(*Spectroscopy scanning Mode*)
IF IsSSMotionMode THEN
	SSMotionMode:=TRUE;
	RegularMotionMode:=FALSE;
ELSE
	SSMotionMode:=FALSE;
	RegularMotionMode:=TRUE;
END_IF
IF	SSMotionMode AND NOT RegularMotionMode THEN
	A_SpectroscopyScanningMotion();
END_IF

(*CheckInputPosVelo*)
A_CheckInputPosVelo();
(*检查光栅读数是否在范围内*)
A_CheckLinearEncoder();

ACTION A_CheckCoupleStatus:
IF NOT btn_PowerOff THEN
	IF st_Power=1 AND st_Couple<>0THEN
		Error:=TRUE;
		ErrorID:=501;
		LeftTopLinMoveIndicator:=0;
		RightTopLinMoveIndicator:=0;
		LeftBottomLinMoveIndicator:=0;
		RightBottomLinMoveIndicator:=0;
		FB_PlcEmergencyStop();
		LED_Error:=TRUE;
		ErrorDescription:='couple stutas error';
	END_IF
END_IF
END_ACTION

ACTION A_CheckInputPosVelo:
//gap posiion
IF UserGapPositionNew<min_UserGapPositionNew OR UserGapPositionNew>max_UserGapPositionNew THEN
	inRange_UserGapPositionNew:=FALSE;
END_IF
IF UserGapPositionNew>=min_UserGapPositionNew AND UserGapPositionNew<=max_UserGapPositionNew THEN
	inRange_UserGapPositionNew:=TRUE;
END_IF
//gap velocity
IF UserGapVelocityNew<min_UserGapVelocityNew OR UserGapVelocityNew>max_UserGapVelocityNew THEN
	inRange_UserGapVelocityNew:=FALSE;
END_IF
IF UserGapVelocityNew>=min_UserGapVelocityNew AND UserGapVelocityNew<=max_UserGapVelocityNew THEN
	inRange_UserGapVelocityNew:=TRUE;
END_IF
//taper position
IF UserTaperPositionNew<min_UserTaperPositionNew OR UserTaperPositionNew>max_UserTaperPositionNew THEN
	inRange_UserTaperPositionNew:=FALSE;
END_IF
IF UserTaperPositionNew>=min_UserTaperPositionNew AND UserTaperPositionNew<=max_UserTaperPositionNew THEN
	inRange_UserTaperPositionNew:=TRUE;
END_IF
//taper velocity
IF UserTaperVelocityNew<min_UserTaperVelocityNew OR UserTaperVelocityNew>max_UserTaperVelocityNew THEN
	inRange_UserTaperVelocityNew:=FALSE;
END_IF
IF UserTaperVelocityNew>=min_UserTaperVelocityNew AND UserTaperVelocityNew<=max_UserTaperVelocityNew THEN
	inRange_UserTaperVelocityNew:=TRUE;
END_IF
//SS Mode
IF SS_StepSize<min_SS_StepSize OR SS_StepSize>max_SS_StepSize THEN
	inRange_SS_StepSize:=FALSE;
END_IF
IF SS_StepSize>=min_SS_StepSize AND SS_StepSize<=max_SS_StepSize THEN
	inRange_SS_StepSize:=TRUE;
END_IF
IF SS_StepNumber<min_SS_StepNumber OR SS_StepNumber>max_SS_StepNumber THEN
	inRange_SS_StepNumber:=FALSE;
END_IF
IF SS_StepNumber>=min_SS_StepNumber AND SS_StepNumber<=max_SS_StepNumber THEN
	inRange_SS_StepNumber:=TRUE;
END_IF
IF SS_StepVelocity<min_SS_StepVelocity OR SS_StepVelocity>max_SS_StepVelocity THEN
	inRange_SS_StepVelocity:=FALSE;
END_IF
IF SS_StepVelocity>=min_SS_StepVelocity AND SS_StepVelocity<=max_SS_StepVelocity THEN
	inRange_SS_StepVelocity:=TRUE;
END_IF
IF StepEachTime_ms<min_StepEachTime_ms OR StepEachTime_ms>max_StepEachTime_ms THEN
	inRange_StepEachTime_ms:=FALSE;
END_IF
IF StepEachTime_ms>=min_StepEachTime_ms AND StepEachTime_ms<=max_StepEachTime_ms THEN
	inRange_StepEachTime_ms:=TRUE;
END_IF
END_ACTION

ACTION A_CheckLinearEncoder:
//如果没有使用光栅、或者光栅参数没设置好，则不检查光栅位置
IF NOT USELinearEncoder OR NOT PositionBiasDone THEN
	RETURN;
END_IF
IF Pos_LeftTopLin <=0 THEN
	ErrorID:=1101;
	Error:=TRUE;
	ErrorDescription:='Pos_LeftTopLin <=0';
	FB_PlcEmergencyStop();
	LED_Error:=TRUE;
END_IF
IF Pos_RightTopLin <=0 THEN
	ErrorID:=1102;
	Error:=TRUE;
	ErrorDescription:='Pos_RightTopLin <=0';
	FB_PlcEmergencyStop();
	LED_Error:=TRUE;
END_IF
IF Pos_LeftBottomLin <=0 THEN
	ErrorID:=1103;
	Error:=TRUE;
	ErrorDescription:='Pos_LeftBottomLin <=0';
	FB_PlcEmergencyStop();
	LED_Error:=TRUE;
END_IF
IF Pos_RightBottomLin <=0 THEN
	ErrorID:=1104;
	Error:=TRUE;
	ErrorDescription:='Pos_RightBottomLin <=0';
	FB_PlcEmergencyStop();
	LED_Error:=TRUE;
END_IF
//
IF Pos_LeftTopLin >UserMode.max_UserGapPositionNew/2 THEN
	ErrorID:=1105;
	Error:=TRUE;
	ErrorDescription:='Pos_LeftTopLin >UserMode.max_UserGapPositionNew';
	FB_PlcEmergencyStop();
	LED_Error:=TRUE;
END_IF
IF Pos_RightTopLin >UserMode.max_UserGapPositionNew/2 THEN
	ErrorID:=1106;
	Error:=TRUE;
	ErrorDescription:='Pos_RightTopLin>UserMode.max_UserGapPositionNew';
	FB_PlcEmergencyStop();
	LED_Error:=TRUE;
END_IF
IF Pos_LeftBottomLin >UserMode.max_UserGapPositionNew/2 THEN
	ErrorID:=1107;
	Error:=TRUE;
	ErrorDescription:='Pos_LeftBottomLin >UserMode.max_UserGapPositionNew';
	FB_PlcEmergencyStop();
	LED_Error:=TRUE;
END_IF
IF Pos_RightBottomLin >UserMode.max_UserGapPositionNew/2 THEN
	ErrorID:=1108;
	Error:=TRUE;
	ErrorDescription:='Pos_RightBottomLin >UserMode.max_UserGapPositionNew';
	FB_PlcEmergencyStop();
	LED_Error:=TRUE;
END_IF

//
IF Pos_LeftTopLin <UserMode.min_UserGapPositionNew/2 THEN
	ErrorID:=1109;
	Error:=TRUE;
	ErrorDescription:='Pos_LeftTopLin <UserMode.min_UserGapPositionNew/2';
	FB_PlcEmergencyStop();
	LED_Error:=TRUE;
END_IF
IF Pos_RightTopLin <UserMode.min_UserGapPositionNew/2 THEN
	ErrorID:=1110;
	Error:=TRUE;
	ErrorDescription:='Pos_RightTopLin<UserMode.min_UserGapPositionNew/2';
	FB_PlcEmergencyStop();
	LED_Error:=TRUE;
END_IF
IF Pos_LeftBottomLin <UserMode.min_UserGapPositionNew/2 THEN
	ErrorID:=1111;
	Error:=TRUE;
	ErrorDescription:='Pos_LeftBottomLin <UserMode.min_UserGapPositionNew';
	FB_PlcEmergencyStop();
	LED_Error:=TRUE;
END_IF
IF Pos_RightBottomLin <UserMode.min_UserGapPositionNew/2 THEN
	ErrorID:=1112;
	Error:=TRUE;
	ErrorDescription:='Pos_RightBottomLin <UserMode.min_UserGapPositionNew';
	FB_PlcEmergencyStop();
	LED_Error:=TRUE;
END_IF
END_ACTION

ACTION A_InitCompensationData:
(*补偿开始*)
IF USE_SingleAxis_Compensation THEN
	//
	//1.目标位置解算
	//
	(*通过补偿表解算四轴目标位置*)
	//左轴位置由Gap定，右轴位置由右gap定。右gap值=左gap+taper。taper模式和非taper模式一样，非taper模式只是一种特例存在
	//左轴目标位置解算
	IF NOT TaperOrNot THEN
		UserTaperPositionNew:=0;
		UserTaperPositionDisplay:=0;
	END_IF
	UserRightGapPositionNew:=UserGapPositionNew+UserTaperPositionNew;
	//左轴目标位置解算
	FOR	i:= 1 TO 17 DO
			IF UserGapPositionNew/2<M_Compensation[i+1].Encoder AND UserGapPositionNew/2>=M_Compensation[i].Encoder THEN
				IF i<>18 THEN
					LeftTopLinPositionNew:=(((UserGapPositionNew/2-M_Compensation[i].Encoder)*(M_Compensation[i+1].LeftTop-M_Compensation[i].LeftTop))
							/(M_Compensation[i+1].Encoder-M_Compensation[i].Encoder))+M_Compensation[i].LeftTop;
					LeftBottomLinPositionNew:=(((UserGapPositionNew/2-M_Compensation[i].Encoder)*(M_Compensation[i+1].LeftBottom-M_Compensation[i].LeftBottom))
							/(M_Compensation[i+1].Encoder-M_Compensation[i].Encoder))+M_Compensation[i].LeftBottom;
					M_CompensationNumber:=i;
					InitCompensationDatasDone:=TRUE;
				ELSIF i=18 AND UserGapPositionNew/2=M_Compensation[i].Encoder THEN		(*Gap=14µÄÌØÊâÇé¿ö*)
					(**)
					LeftTopLinPositionNew:=M_Compensation[i].LeftTop;
					LeftBottomLinPositionNew:=M_Compensation[i].LeftBottom;
					M_CompensationNumber:=i;
					InitCompensationDatasDone:=TRUE;
				ELSE
					LeftTopLinPositionNew:=UserGapPositionNew/2;
					LeftBottomLinPositionNew:=UserGapPositionNew/2;
					M_CompensationNumber:=i;
					InitCompensationDatasDone:=TRUE;
				END_IF
			END_IF
	END_FOR
	//右轴目标位置解算
	FOR	j:= 1 TO 17 DO
		IF UserRightGapPositionNew/2<M_Compensation[j+1].Encoder AND UserRightGapPositionNew/2>=M_Compensation[j].Encoder THEN
			IF j<>18 THEN
				RightTopLinPositionNew:=(((UserRightGapPositionNew/2-M_Compensation[j].Encoder)*(M_Compensation[j+1].RightTop-M_Compensation[j].RightTop))
						/(M_Compensation[j+1].Encoder-M_Compensation[j].Encoder))+M_Compensation[j].RightTop;
				RightBottomLinPositionNew:=(((UserRightGapPositionNew/2-M_Compensation[j].Encoder)*(M_Compensation[j+1].RightBottom-M_Compensation[j].RightBottom))
						/(M_Compensation[j+1].Encoder-M_Compensation[j].Encoder))+M_Compensation[j].RightBottom;
				M_CompensationNumber:=j;
				InitCompensationDatasDone:=TRUE;
			ELSIF j=18 AND UserRightGapPositionNew/2=M_Compensation[i].Encoder THEN		(*Gap=14µÄÌØÊâÇé¿ö*)
				(**)
				RightTopLinPositionNew:=M_Compensation[i].RightTop;
				RightBottomLinPositionNew:=M_Compensation[i].RightBottom;
				M_CompensationNumber:=j;
				InitCompensationDatasDone:=TRUE;
			ELSE
				RightTopLinPositionNew:=UserGapPositionNew/2;
				RightBottomLinPositionNew:=UserGapPositionNew/2;
				M_CompensationNumber:=j;
				InitCompensationDatasDone:=TRUE;
			END_IF
		END_IF
	END_FOR
	//
	//2.不论taper还是非taper模式，左轴gap都有左轴发推算，右轴gap由右轴反推算。taper为右gap-左gap
	//
	//左轴显示位置反结算
	FOR k:= 1 TO 17 DO
			IF Pos_LeftTopLin<M_Compensation[k+1].LeftTop AND Pos_LeftTopLin>=M_Compensation[k].LeftTop THEN
				UserGapPositionDisplay_FromLeftTop:=2*(((Pos_LeftTopLin-M_Compensation[k].LeftTop)*(M_Compensation[k+1].Encoder-M_Compensation[k].Encoder))
											/(M_Compensation[k+1].LeftTop-M_Compensation[k].LeftTop)+M_Compensation[k].Encoder);
				UserGapPositionDisplay_FromLeftBottom:=2*(((Pos_LeftBottomLin-M_Compensation[k].LeftBottom)*(M_Compensation[k+1].Encoder-M_Compensation[k].Encoder))
											/(M_Compensation[k+1].LeftBottom-M_Compensation[k].LeftBottom)+M_Compensation[k].Encoder);
				UserGapPositionDisplay:=DINT_TO_LREAL(LREAL_TO_DINT(((UserGapPositionDisplay_FromLeftTop+UserGapPositionDisplay_FromLeftBottom)/2)*100000))/100000;
			END_IF
	END_FOR
	//右轴显示位置反结算
	FOR m:= 1 TO 17 DO
			IF Pos_RightTopLin<M_Compensation[m+1].RightTop AND Pos_RightTopLin>=M_Compensation[m].RightTop THEN
				UserRightGapPositionDisplay_FromRightTop:=2*(((Pos_RightTopLin-M_Compensation[m].RightTop)*(M_Compensation[m+1].Encoder-M_Compensation[m].Encoder))
											/(M_Compensation[m+1].RightTop-M_Compensation[m].RightTop)+M_Compensation[m].Encoder);
				UserRightGapPositionDisplay_FromRightBottom:=2*(((Pos_RightBottomLin-M_Compensation[m].RightBottom)*(M_Compensation[m+1].Encoder-M_Compensation[m].Encoder))
											/(M_Compensation[m+1].RightBottom-M_Compensation[m].RightBottom)+M_Compensation[m].Encoder);
				UserRightGapPositionDisplay:=(UserRightGapPositionDisplay_FromRightTop+UserRightGapPositionDisplay_FromRightBottom)/2;
			END_IF
	END_FOR
	IF TaperOrNot THEN
		UserTaperPositionDisplay:=DINT_TO_LREAL(LREAL_TO_DINT((UserRightGapPositionDisplay-UserGapPositionDisplay)*100000))/100000;
	END_IF
END_IF
(*速度可以不用解算，直接用即可*)
LeftTopLinVelocityDisplay:=Velo_LeftTopLin;
RightTopLinVelocityDisplay:=Velo_RightTopLin;
LeftBottomLinVelocityDisplay:=Velo_LeftBottomLin;
RightBottomLinVelocityDisplay:=Velo_RightBottomLin;
//Gap velocity
UserGapVelocityDisplay:=DINT_TO_LREAL(LREAL_TO_DINT(((LeftTopLinVelocityDisplay+RightTopLinVelocityDisplay+
	LeftBottomLinVelocityDisplay+RightBottomLinVelocityDisplay)/2)*100000))/100000;
END_ACTION

ACTION A_MonitoringAllAxis:
(****************************************************************
NAME:			A_MonitoringAllAxis
DATA:			2018.1.9
VERSION:		1.0.0
DESCRIPTION:	
				Ã¿´ÎÑ­»·¾ùÖ´ÐÐÖáÎ»ÖÃºÍÖáÔË¶¯µÄ¼ì²é
				2.4Öá¹âÕ¤³ßÎ»ÖÃ¡¢ËÙ¶È¶Ô±È¼ì²é
HISTORY:
				2017.1.9		NEW

***************************************************************)

(*************************************************************************************2.4Öá¹âÕ¤³ßÎ»ÖÃ¡¢ËÙ¶È¶Ô±È¼ì²é**********************************************************************)
IF  st_Power<>0 THEN
CASE moni_State OF
(*Top Î»ÖÃºÍËÙ¶È±È¶Ô*)
0:
		//实际(*Position*)
		(*Top*)
		Diff_UserTopPos_actual:=ABS(Pos_leftTopLin-Pos_RightTopLin);
		(*Bottom*)
		Diff_UserBottomPos_actual:=ABS(Pos_LeftBottomLin-Pos_RightBottomLin);
		(*Left*)
		Diff_UserLeftPos_actual:=ABS(Pos_LeftTopLin-Pos_LeftBottomLin);
		(*Right*)
		Diff_UserRightPos_actual:=ABS(Pos_RightTopLin-Pos_RightBottomLin);
		(*Velocity*)
		(*Top*)
		Diff_UserTopVelo_actual:=ABS(Velo_leftTopLin-Velo_RightTopLin);
		(*Bottom*)
		Diff_UserBottomVelo_actual:=ABS(Velo_LeftBottomLin-Velo_RightBottomLin);
		(*Left*)
		Diff_UserLeftVelo_actual:=ABS(Velo_LeftTopLin-Velo_LeftBottomLin);
		(*Right*)
		Diff_UserRightVelo_actual:=ABS(Velo_RightTopLin-Velo_RightBottomLin);
		//阈值
		Threshold_UserTopPos_PLC:=Threshold_UserTopPos+UserTaperPositionDisplay;//Top位置误差=gap运动细微误差+目标taper位置
		Threshold_UserTopVelo_PLC:=Threshold_UserTopVelo+ABS(UserGapVelocityDisplay);//Top速度误差=gap运动细微误差+gap目标速度。因为可能出现一个轴运动完了，另一个轴还在运动的情况
		Threshold_UserBottomPos_PLC:=Threshold_UserBottomPos+UserTaperPositionDisplay;//Bottom同上
		Threshold_UserBottomVelo_PLC:=Threshold_UserBottomVelo+ABS(UserGapVelocityDisplay);//Bottom同上
		Threshold_UserLeftPos_PLC:=Threshold_UserLeftPos+UserTaperPositionDisplay;
		Threshold_UserLeftVelo_PLC:=Threshold_UserLeftVelo+ABS(UserGapVelocityDisplay);
		Threshold_UserRightPos_PLC:=Threshold_UserRightPos+UserTaperPositionDisplay;
		Threshold_UserRightVelo_PLC:=Threshold_UserRightVelo+ABS(UserGapVelocityDisplay);
		//比较
		IF Diff_UserTopPos_actual >Threshold_UserTopPos_PLC THEN
				Error:=TRUE;
				ErrorID:=601;
				ErrorDescription:='Diff_UserTopPos_actual >Threshold_UserTopPos_PLC';
				moni_State:=-100;
		ELSIF Diff_UserTopVelo_actual>Threshold_UserTopVelo_PLC  THEN
				Error:=TRUE;
				ErrorID:=602;
				ErrorDescription:='Diff_UserTopVelo_actual>Threshold_UserTopVelo_PLC';
				moni_State:=-100;
		(*Bottom Î»ÖÃºÍËÙ¶È±È¶Ô*)
		ELSIF Diff_UserBottomPos_actual>Threshold_UserBottomPos_PLC THEN
				Error:=TRUE;
				ErrorID:=603;
				ErrorDescription:='Diff_UserBottomPos_actual>Threshold_UserBottomPos_PLC';
				moni_State:=-100;
		ELSIF Diff_UserBottomVelo_actual>Threshold_UserBottomVelo_PLC  THEN
				Error:=TRUE;
				ErrorID:=604;
				ErrorDescription:='Diff_UserBottomVelo_actual>Threshold_UserBottomVelo_PLC';
				moni_State:=-100;
		(*Left Î»ÖÃºÍËÙ¶È±È¶Ô*)
		ELSIF Diff_UserLeftPos_actual>Threshold_UserLeftPos_PLC  THEN
				Error:=TRUE;
				ErrorID:=605;
				ErrorDescription:='Diff_UserLeftPos_actual>Threshold_UserLeftPos_PLC';
				moni_State:=-100;
		ELSIF  Diff_UserLeftVelo_actual>Threshold_UserLeftVelo_PLC THEN
				Error:=TRUE;
				ErrorID:=606;
				ErrorDescription:='Diff_UserLeftVelo_actual>Threshold_UserLeftVelo_PLC';
				moni_State:=-100;
		(*Right Î»ÖÃºÍËÙ¶È±È¶Ô*)
		ELSIF Diff_UserRightPos_actual>Threshold_UserRightPos_PLC  THEN
				Error:=TRUE;
				ErrorID:=607;
				ErrorDescription:='Diff_UserRightPos_actual>Threshold_UserRightPos_PLC';
				moni_State:=-100;
		ELSIF  Diff_UserRightVelo_actual>Threshold_UserRightVelo_PLC THEN
				Error:=TRUE;
				ErrorID:=608;
				ErrorDescription:='Diff_UserRightVelo_actual>Threshold_UserRightVelo_PLC';
				moni_State:=-100;
		END_IF
-100:
		btn_UserGapStop:=TRUE;
		FB_PlcEmergencyStop();
		Error:=TRUE;
		LED_Error:=TRUE;
END_CASE
END_IF
END_ACTION

ACTION A_PowerOff:
CASE d_state OF
		0:(*PowerOff*)
			FB_Power(Off:=TRUE);
				d_state:=1;
		1:
			IF NOT FB_power.OffStatus THEN
				d_state:=1;
			ELSE
				d_state:=88;
			END_IF
		88:(*ResetAllState*)
			btn_PowerOn:=FALSE;
			btn_UserGapMove:=FALSE;
			btn_UserGapStop:=FALSE;
			LeftTopLinMoveIndicator:=0;
			RightTopLinMoveIndicator:=0;
			LeftBottomLinMoveIndicator:=0;
			RightBottomLinMoveIndicator:=0;
			fb_ton1.IN:=FALSE;
			fb_ton2.IN:=FALSE;
			fb_ton3.IN:=FALSE;
			State:=0;
			Busy:=FALSE;
			InitPowerDone:=FALSE;
			InitCompensationDatasDone:=FALSE;
			Error:=FALSE;
			ErrorID:=0;
			m_state:=0;
			n_state:=0;
			s_state:=0;
			btn_PowerOff:=FALSE;
			d_state:=0;
			Led_Run:=FALSE;
			Led_Error:=FALSE;
			moni_State:=0;
			i:=0;
END_CASE
END_ACTION

ACTION A_PowerOn:
(****************************************************************
NAME:			A_PowerOn
DATA:			2018.1.9
VERSION:		1.0.0
DESCRIPTION:	
				ÉÏµãÃüÁîºó£¬Ë³ÐòÖ´ÐÐ£º
				1.FB_PowerOn
				·µ»ØÖ´ÐÐÊÇ·ñ³É¹¦
HISTORY:
				2019.1.9		NEW

***************************************************************)
fb_ton3(PT:=t#0.5s);
CASE State OF
	0:	(*FB_Power_On*)
		FB_Power(On:=TRUE);
		fb_ton3.IN:=TRUE;
		State:=1;
	1:	(*wait*)
		FB_power();
		IF NOT FB_power.OnStatus THEN		(*FB_Power_OnÃ»ÓÐÖ´ÐÐÍê£¬wait£¬³¬Ê±FB Error*)
			IF NOT fb_ton3.Q THEN
				State:=1;
			ELSE
				ErrorID:=1;
				State:=99;
			END_IF
		ELSE
			State:=88;
		END_IF
	88:	(*All Done*)
		btn_PowerOn:=FALSE;
		State:=0;
		Error:=FALSE;
		ErrorID:=0;
		Busy:=FALSE;
		InitPowerDone:=TRUE;
		FB_power.On:=FALSE;
		fb_ton3.IN:=FALSE;
		LED_Error:=FALSE;
	99:
		Error:=TRUE;
		//ErrorID:=701;
		//ErrorDescription:='power on error';		
		btn_PowerOn:=FALSE;
		State:=99;
		Busy:=FALSE;
		InitPowerDone:=FALSE;
		fb_ton3.IN:=FALSE;
		LED_Error:=TRUE;
END_CASE
END_ACTION

ACTION A_RegularMotion:
(*输入保护*)
IF btn_UserGapMove AND NOT SSMotionMode AND RegularMotionMode THEN
	IF NOT inRange_UserGapPositionNew THEN
		btn_UserGapStop:=TRUE;
		btn_UserGapMove:=FALSE;
		Error:=TRUE;
		ErrorId:=801;
		ErrorDescription:='target Gap position out of range,please check';
		RETURN;
	ELSE
		btn_UserGapStop:=FALSE;
		Error:=FALSE;
		ErrorId:=0;
		ErrorDescription:='';	
	END_IF
	IF NOT inRange_UserGapVelocityNew THEN
		btn_UserGapStop:=TRUE;
		btn_UserGapMove:=FALSE;
		Error:=TRUE;
		ErrorId:=802;
		ErrorDescription:='target Gap velocity out of range,please check';
		RETURN;
	ELSE
		btn_UserGapStop:=FALSE;
		Error:=FALSE;
		ErrorId:=0;
		ErrorDescription:='';
	END_IF
	IF NOT inRange_UserTaperPositionNew THEN
		btn_UserGapStop:=TRUE;
		btn_UserGapMove:=FALSE;
		Error:=TRUE;
		ErrorId:=803;
		ErrorDescription:='target Taper Position out of range,please check';
		RETURN;
	ELSE
		btn_UserGapStop:=FALSE;
		Error:=FALSE;
		ErrorId:=0;
		ErrorDescription:='';
	END_IF
	IF NOT inRange_UserTaperVelocityNew THEN
		btn_UserGapStop:=TRUE;
		btn_UserGapMove:=FALSE;
		Error:=TRUE;
		ErrorId:=804;
		ErrorDescription:='target Taper velocity out of range,please check';
		RETURN;
	ELSE
		btn_UserGapStop:=FALSE;
		Error:=FALSE;
		ErrorId:=0;
		ErrorDescription:='';
	END_IF
END_IF
(*若GAP将有变化，首先检测TAPER是否超出阈值，若超出，则报错，提示必须先将TAPER回归到0，才可以改变GAP*)
IF ABS(UserGapPositionNew-UserGapPositionDisplay)>Threshold_GapChangeFlag AND btn_UserGapMove THEN
	IF UserTaperPositionDisplay>Threshold_TaperChangeFlag THEN
		btn_UserGapStop:=TRUE;
		btn_UserGapMove:=FALSE;
		Error:=TRUE;
		ErrorId:=809;
		ErrorDescription:='Please Move Taper to zero first before move gap';
		RETURN;
	END_IF
END_IF
(*Taper和gap连锁限制性保护。比如11mm时候如果taper，入口端gap变小，会有压真空盒的问题。设置保护*)
IF UserGapPositionNew-TaperAndGapSafetyfactor*0.41*UserTaperPositionNew<=min_UserGapPositionNew AND btn_UserGapMove THEN
		btn_UserGapStop:=TRUE;
		btn_UserGapMove:=FALSE;
		Error:=TRUE;
		ErrorId:=810;
		ErrorDescription:='Target taper is too big at current Gap';
		RETURN;
END_IF
(*分别比较四轴目标位置与当前位置的差，如果目标位置比当前位置低，则需要运动到更低-回程差一半；再运动至最终目标位置*)
(*
IF LeftTopLinPositionNew-Pos_LeftTopLin>LEDriftErrorThreshold AND RightTopLinPositionNew-Pos_RightTopLin>LEDriftErrorThreshold 
	AND LeftBottomLinPositionNew-Pos_LeftBottomLin>LEDriftErrorThreshold AND RightBottomLinPositionNew-Pos_RightBottomLin>LEDriftErrorThreshold THEN
		TargetPosLessThanCurrentPos:=FALSE;//四轴目标位置都大于当前位置，直接走到目标位置即可，不需要先走到考虑回城误差的临时位置
END_IF
*)
//只在m=和n=0的时候判断，否则会出现一些BUG，比如往大间隙开时，运动到位后m不能回到0.
IF m_state=0 AND n_state=0 THEN
		TargetPosLessThanCurrentPos:=FALSE;
	IF LeftTopLinPositionNew-Pos_LeftTopLin<-LEDriftErrorThreshold THEN
			TargetPosLessThanCurrentPos:=TRUE;
			TargetLTPosLessThanCurrentLTPos:=TRUE;
	ELSE
				TargetLTPosLessThanCurrentLTPos:=FALSE;
	END_IF
	IF RightTopLinPositionNew-Pos_RightTopLin<-LEDriftErrorThreshold THEN
			TargetPosLessThanCurrentPos:=TRUE;
			TargetRTPosLessThanCurrentRTPos:=TRUE;
	ELSE
			TargetRTPosLessThanCurrentRTPos:=FALSE;
	END_IF
	IF LeftBottomLinPositionNew-Pos_LeftBottomLin<-LEDriftErrorThreshold THEN
			TargetPosLessThanCurrentPos:=TRUE;
			TargetLBPosLessThanCurrentLBPos:=TRUE;
	ELSE
			TargetLBPosLessThanCurrentLBPos:=FALSE;
	END_IF
	IF RightBottomLinPositionNew-Pos_RightBottomLin<-LEDriftErrorThreshold THEN
			TargetPosLessThanCurrentPos:=TRUE;
			TargetRBPosLessThanCurrentRBPos:=TRUE;
	ELSE
			TargetRBPosLessThanCurrentRBPos:=FALSE;
	END_IF
END_IF

(*Move*)
IF InitPowerDone AND InitCompensationDatasDone THEN
	//IF btn_UserGapMove THEN
		(*四轴目标位置都大于当前位置，直接走到目标位置即可，不需要先走到考虑回城误差的临时位置*)
		IF NOT TargetPosLessThanCurrentPos AND NOT HysteresisMoving THEN
			CASE m_state OF
				0:
					FB_Move.Mode:=5;						//1.gap;2.single;3.taper;4.debug;5.BCGap&UserMode
					FB_Move.CoupleState:=st_Couple;			
					FB_Move.PowerState:=st_Power;							
					FB_Move.BCLeftTopPosition:=LeftTopLinPositionNew;
					FB_Move.BCLeftTopVelocity:=UserGapVelocityNew/2;
					FB_Move.BCRightTopPosition:=RightTopLinPositionNew;
					FB_Move.BCRightTopVelocity:=UserGapVelocityNew/2;
					FB_Move.BCLeftBottomPosition:=LeftBottomLinPositionNew;
					FB_Move.BCLeftBottomVelocity:=UserGapVelocityNew/2;
					FB_Move.BCRightBottomPosition:=RightBottomLinPositionNew;
					FB_Move.BCRightBottomVelocity:=UserGapVelocityNew/2;		
					IF btn_UserGapMove THEN
						FB_Move.BCGapMove:=TRUE;
						m_state:=1;
						FB_Move();
					END_IF
				1:
					btn_UserGapMove:=FALSE;
					FB_Move();
					IF NOT FB_Move.BCGapDone THEN			(*ÔË¶¯Î´Íê³É£¬Ñ­»·*)
						Led_Run:=TRUE;
						m_state:=1;
					ELSE									(*ÔË¶¯Íê³É£¬ÏÂÒ»²½*)
						m_state:=88;
					END_IF
				88:
					btn_UserGapMove:=FALSE;					(*×´Ì¬»Ö¸´*)
					Led_Run:=FALSE;
					m_state:=0;
			END_CASE
		(*四轴有目标位置小于当前位置，先走到临时位置，再走到目标位置*)
		ELSE
			CASE n_state OF
				0:
					FB_Move.Mode:=5;						//1.gap;2.single;3.taper;4.debug;5.BCGap&UserMode;5:userMode_2
					FB_Move.CoupleState:=st_Couple;			
					FB_Move.PowerState:=st_Power;			
					
					//
					IF TargetLTPosLessThanCurrentLTPos THEN			
						FB_Move.BCLeftTopPosition:=LeftTopLinPositionNew-HysteresisError/2;
					ELSE
						FB_Move.BCLeftTopPosition:=LeftTopLinPositionNew;	
					END_IF
					//
					IF TargetRTPosLessThanCurrentRTPos THEN 
						FB_Move.BCRightTopPosition:=RightTopLinPositionNew-HysteresisError/2;
					ELSE					
						FB_Move.BCRightTopPosition:=RightTopLinPositionNew;
					END_IF
					//
					IF TargetLBPosLessThanCurrentLBPos THEN
						FB_Move.BCLeftBottomPosition:=LeftBottomLinPositionNew-HysteresisError/2;
					ELSE
						FB_Move.BCLeftBottomPosition:=LeftBottomLinPositionNew;
					END_IF
					//
					IF TargetRBPosLessThanCurrentRBPos THEN
						FB_Move.BCRightBottomPosition:=RightBottomLinPositionNew-HysteresisError/2;
					ELSE
						FB_Move.BCRightBottomPosition:=RightBottomLinPositionNew;
					END_IF					
					//
					FB_Move.BCLeftTopVelocity:=UserGapVelocityNew/2;
					FB_Move.BCRightTopVelocity:=UserGapVelocityNew/2;
					FB_Move.BCLeftBottomVelocity:=UserGapVelocityNew/2;
					FB_Move.BCRightBottomVelocity:=UserGapVelocityNew/2;
						
					IF btn_UserGapMove THEN							
						n_state:=1;
						FB_Move.BCGapMove:=TRUE;
						FB_Move();
						HysteresisMoving:=TRUE;
					END_IF
				1:
					btn_UserGapMove:=FALSE;
					FB_Move();
					IF NOT FB_Move.BCGapDone THEN			(*还未运动到位置,运动过程中*)
						Led_Run:=TRUE;
						n_state:=1;
					ELSE									
						n_state:=2;							(*转到下一步，运动到最终位置*)
						FB_Move.BCGapMove:=FALSE;
						//Led_Run:=FALSE;
					END_IF
					(*
					IF NOT Unreach_LS_Bottom THEN
						n_state:=2;							(*在运动过程中如果碰到下限位，则也转到下一步，运动到最终位置*)
						FB_Move.BCGapMove_2:=FALSE;
						FB_Move.BCGapReset_2:=TRUE;
					END_IF
					*)
				2:
					FB_Move.BCGapReset:=FALSE;
					FB_Move.Mode:=5;						//1.gap;2.single;3.taper;4.debug;5.BCGap&UserMode
					FB_Move.CoupleState:=st_Couple;			
					FB_Move.PowerState:=st_Power;			
					FB_Move.BCGapMove:=TRUE;
					//直接走到目标位置，已经走到位置的，可以继续下命令，只不过它不在走了而已
					FB_Move.BCLeftTopPosition:=LeftTopLinPositionNew;	
					FB_Move.BCRightTopPosition:=RightTopLinPositionNew;
					FB_Move.BCLeftBottomPosition:=LeftBottomLinPositionNew;
					FB_Move.BCRightBottomPosition:=RightBottomLinPositionNew;
					//
					FB_Move.BCLeftTopVelocity:=UserGapVelocityNew/2;
					FB_Move.BCRightTopVelocity:=UserGapVelocityNew/2;
					FB_Move.BCLeftBottomVelocity:=UserGapVelocityNew/2;
					FB_Move.BCRightBottomVelocity:=UserGapVelocityNew/2;
					FB_Move();							
					n_state:=3;
				3:
					FB_Move();
					IF NOT FB_Move.BCGapDone THEN			(*还未运动到位置,运动过程中*)
						Led_Run:=TRUE;
						n_state:=3;
					ELSE									
						n_state:=88;							(*运动到了最终位置*)
					END_IF
					(*
					IF NOT Unreach_LS_Bottom THEN
						n_state:=88;							(*在运动过程中如果碰到下限位，则也转到下一步，运动到最终位置*)
						FB_Move.BCGapMove_2:=FALSE;
					END_IF
					*)
				88:
					btn_UserGapMove:=FALSE;					
					Led_Run:=FALSE;
					n_state:=0;
					HysteresisMoving:=FALSE;
			END_CASE
		END_IF
	//END_IF
END_IF

IF btn_UserGapStop THEN
	FB_Move.BCGapReset:=TRUE;							(*¸øÔË¶¯FB¸øÍ£Ö¹ÐÅºÅ£¬Ê¹FB_Move×´Ì¬»Ö¸´*)
	FB_Move();											(*Æô¶¯FB_Move*)
	btn_UserGapMove:=FALSE;								(*btn_GapMove:=FALSE*)
	m_state:=0;	
	n_state:=0;										(*m_state:=0;*)
	CASE s_state OF
			0:
				FB_Stop.Mode:=5;							(*1£ºgapÄ£Ê½£»2£ºµ¥ÁºÄ£Ê½£»3£ºtaperÄ£Ê½£»4£ºDebugÄ£Ê½£»5£ºBCGapÄ£Ê½*)
				FB_Stop.CoupleState:=st_Couple;			(*ñîºÏ×´Ì¬ÊäÈë*)
				FB_Stop.PowerState:=st_Power;				(*µçÔ´×´Ì¬ÊäÈë*)
				FB_Stop.BCGapStop:=TRUE;				(*Execute TRUE*)
				FB_Stop();								(*Æô¶¯FB*)
				s_state:=1;
			1:
				FB_Stop();
				IF NOT FB_Stop.BCGapDone THEN			(*Í£Ö¹Î´Íê³É£¬Ñ­»·*)
					s_state:=1;
				ELSE									(*Í£Ö¹Íê³É£¬ÏÂÒ»²½*)
					s_state:=88;
				END_IF
			88:
				btn_UserGapStop:=FALSE;						(*»Ö¸´×´Ì¬*)
				FB_Move.BCGapReset:=FALSE;				(*ÔËÐÐFB*)
				s_state:=0;
		END_CASE
END_IF

(*触发限位开关后，相当于点击了Stop按钮*)
FTrig_ReachLS(CLK:=Unreach_LS_Top AND Unreach_LS_Bottom);
IF FTrig_ReachLS.Q THEN
	btn_UserGapStop:=TRUE;
END_IF
END_ACTION

ACTION A_SpectroscopyScanningMotion:
(*输入保护*)
IF SS_Move AND SSMotionMode AND NOT RegularMotionMode THEN
	IF NOT inRange_SS_StepSize THEN
		SS_Stop:=TRUE;
		SS_Move:=FALSE;
		Error:=TRUE;
		ErrorId:=805;
		ErrorDescription:='target StepSize out of range,please check';
		RETURN;
	ELSE
		SS_Stop:=FALSE;
		Error:=FALSE;
		ErrorId:=0;
		ErrorDescription:='';	
	END_IF
	//
	IF NOT inRange_SS_StepNumber THEN
		SS_Stop:=TRUE;
		SS_Move:=FALSE;
		Error:=TRUE;
		ErrorId:=806;
		ErrorDescription:='target StepNumber out of range,please check';
		RETURN;
	ELSE
		SS_Stop:=FALSE;
		Error:=FALSE;
		ErrorId:=0;
		ErrorDescription:='';	
	END_IF
	IF NOT inRange_SS_StepVelocity THEN
		SS_Stop:=TRUE;
		SS_Move:=FALSE;
		Error:=TRUE;
		ErrorId:=807;
		ErrorDescription:='target StepVelocity out of range,please check';
		RETURN;
	ELSE
		SS_Stop:=FALSE;
		Error:=FALSE;
		ErrorId:=0;
		ErrorDescription:='';	
	END_IF
	IF NOT inRange_StepEachTime_ms THEN
		SS_Stop:=TRUE;
		SS_Move:=FALSE;
		Error:=TRUE;
		ErrorId:=808;
		ErrorDescription:='target StepEachTime_ms out of range,please check';
		RETURN;
	ELSE
		SS_Stop:=FALSE;
		Error:=FALSE;
		ErrorId:=0;
		ErrorDescription:='';	
	END_IF
END_IF
(*单步时长转换*)
StepEachTime:=INT_TO_TIME(StepEachTime_ms);
SS_TON(PT:=StepEachTime);
(*上升沿触发，初始SS位置=当前磁间隙*)
RTRG_SS_StartPositionDisplay(CLK:=SS_Move);
IF RTRG_SS_StartPositionDisplay.Q THEN
	SS_StartPositionDisplay:=UserGapPositionDisplay;
	SS_InitStartPositionDone:=TRUE;
END_IF
(*SS主程序*)
IF InitPowerDone AND InitCompensationDatasDone AND SS_Move AND SS_InitStartPositionDone THEN
	CASE SS_MoveState OF
		0:
				//UserGapPositionNew:=UserGapPositionDisplay+SS_StepSize;
				UserGapPositionNew:=SS_StartPositionDisplay+SS_StepSize*(SS_currentStep+1);
				A_InitCompensationData();
				FB_Move.Mode:=5;						//1.gap;2.single;3.taper;4.debug;5.BCGap&UserMode
				FB_Move.CoupleState:=st_Couple;			
				FB_Move.PowerState:=st_Power;							
				FB_Move.BCLeftTopPosition:=LeftTopLinPositionNew;
				FB_Move.BCLeftTopVelocity:=UserGapVelocityNew/2;
				FB_Move.BCRightTopPosition:=RightTopLinPositionNew;
				FB_Move.BCRightTopVelocity:=UserGapVelocityNew/2;
				FB_Move.BCLeftBottomPosition:=LeftBottomLinPositionNew;
				FB_Move.BCLeftBottomVelocity:=UserGapVelocityNew/2;
				FB_Move.BCRightBottomPosition:=RightBottomLinPositionNew;
				FB_Move.BCRightBottomVelocity:=UserGapVelocityNew/2;		
				FB_Move.BCGapMove:=TRUE;
				FB_Move();
				SS_MoveState:=1;
		1:
				SS_TON.IN:=TRUE;
				FB_Move();
				IF FB_Move.GapMoving AND NOT SS_TimeCountBegin THEN
					SS_StepSystemTime_Begin[SS_currentStep]:=F_GetSysTime();
					SS_TimeCountBegin:=TRUE;
				END_IF
				IF NOT FB_Move.BCGapDone THEN			
					Led_Run:=TRUE;
					SS_MoveState:=1;
				ELSE									
					SS_MoveState:=66;
					SS_StepSystemTime_End[SS_currentStep]:=F_GetSysTime();
					SS_StepCountTime[SS_currentStep]:=SS_StepSystemTime_End[SS_currentStep]-SS_StepSystemTime_Begin[SS_currentStep];
					SS_TimeCountBegin:=FALSE;
				END_IF
		66:
				SS_currentStep:=SS_currentStep+1;			
				Led_Run:=FALSE;
				IF SS_currentStep=SS_StepNumber THEN								
					SS_MoveState:=88;
				END_IF
				IF SS_currentStep<SS_StepNumber THEN
					SS_MoveState:=77;
				END_IF
		77://等待单步时长够
				IF SS_TON.Q THEN
					SS_TON.IN:=FALSE;
					SS_MoveState:=0;
				END_IF
		88:
				SS_TON.IN:=FALSE;
				SS_Move:=FALSE;	
				Led_Run:=FALSE;
				SS_MoveState:=0;
				SS_currentStep:=0;
				SS_InitStartPositionDone:=FALSE;
				//SS_StepSystemTime[SS_StepNumber]:=F_GetSysTime();
	END_CASE
END_IF
(*获取每一步耗时*)
//FOR	m:= 0 TO SS_StepNumber DO
//	SS_StepCountTime[m]:=(SS_StepSystemTime_End[m]-SS_StepSystemTime_Begin[m]);
//END_FOR

(*STOP*)
IF SS_Stop THEN
	FB_Move.BCGapReset:=TRUE;							(*¸øÔË¶¯FB¸øÍ£Ö¹ÐÅºÅ£¬Ê¹FB_Move×´Ì¬»Ö¸´*)
	FB_Move();											(*Æô¶¯FB_Move*)
	SS_Move:=FALSE;								(*btn_GapMove:=FALSE*)
	SS_MoveState:=0;										(*m_state:=0;*)
	CASE SS_StopState OF
			0:
				FB_Stop.Mode:=5;							(*1£ºgapÄ£Ê½£»2£ºµ¥ÁºÄ£Ê½£»3£ºtaperÄ£Ê½£»4£ºDebugÄ£Ê½£»5£ºBCGapÄ£Ê½*)
				FB_Stop.CoupleState:=st_Couple;			(*ñîºÏ×´Ì¬ÊäÈë*)
				FB_Stop.PowerState:=st_Power;				(*µçÔ´×´Ì¬ÊäÈë*)
				FB_Stop.BCGapStop:=TRUE;				(*Execute TRUE*)
				FB_Stop();								(*Æô¶¯FB*)
				SS_StopState:=1;
			1:
				FB_Stop();
				IF NOT FB_Stop.BCGapDone THEN			(*Í£Ö¹Î´Íê³É£¬Ñ­»·*)
					SS_StopState:=1;
				ELSE									(*Í£Ö¹Íê³É£¬ÏÂÒ»²½*)
					SS_StopState:=88;
				END_IF
			88:
				SS_Stop:=FALSE;						(*»Ö¸´×´Ì¬*)
				FB_Move.BCGapReset:=FALSE;				(*ÔËÐÐFB*)
				SS_StopState:=0;
		END_CASE
END_IF

(*触发限位开关后，相当于点击了Stop按钮*)
FTrig_ReachLS(CLK:=Unreach_LS_Top AND Unreach_LS_Bottom);
IF FTrig_ReachLS.Q THEN
	SS_Stop:=TRUE;
END_IF
END_ACTION

END_PROGRAM

// ---- POUs/0.UserMode/F_GetSysTime.TcPOU
FUNCTION F_GetSysTime : ULINT
VAR_INPUT
END_VAR
VAR
	GetSystemTime:GETSYSTEMTIME;
END_VAR

GetSystemTime(timeLoDW=>,timeHiDW=>);
F_GetSysTime:=UDINT_TO_ULINT(GetSystemTime.timeHiDW)*4294967296+UDINT_TO_ULINT(GetSystemTime.timeLoDW)/10000;

END_FUNCTION

// ---- POUs/MainPRG/FB_CheckCoupleStatus.TcPOU
(****************************************************************
NAME:			FB_CheckCoupleStatus
DATA:			2017.2.17
VERSION:		1.0.0
DESCRIPTION:	FB_CheckCoupleStatus
HISTORY:
				2017.2.17		NEW

***************************************************************)
FUNCTION_BLOCK FB_CheckCoupleStatus
VAR_INPUT
	Check:BOOL;
END_VAR
VAR_OUTPUT
	CoupleState:DINT;
	FbID:DINT:=1001;
	Busy:BOOL;
	Error:BOOL;
	ErrorID:DINT;
END_VAR
VAR
END_VAR

IF Check THEN
	Busy:=TRUE;
	IF LeftTopLin.NcToPlc.CoupleState=1 AND RightTopLin.NcToPlc.CoupleState=3
		AND LeftBottomLin.NcToPlc.CoupleState=1 AND RightBottomLin.NcToPlc.CoupleState=3 THEN
		CoupleState:=1;
	ELSIF LeftTopLin.NcToPlc.CoupleState=0 AND RightTopLin.NcToPlc.CoupleState=0
		AND LeftBottomLin.NcToPlc.CoupleState=0 AND RightBottomLin.NcToPlc.CoupleState=0 THEN
		CoupleState:=0;
	ELSE
		CoupleState:=-100;
		Error:=TRUE;
		ErrorID:=-100;
		FB_PlcEmergencyStop();
	END_IF
END_IF

END_FUNCTION_BLOCK

// ---- POUs/RS232/BackgroundEL.TcPOU
PROGRAM BackgroundEL
VAR
	fbEL6001Ctrl		: SerialLineControl;
	bEL6001CtrlError	: BOOL;
	eEL6001CtrlErrorID	: ComError_t;
	(* 	I/O variables for a EL6001 terminal*)
	stIn_EL6001 AT %I*	: KL6inData22B;	(* linked to the EL6001 in the TwinCAT System Manager *)
	stOut_EL6001 AT %Q*	: KL6outData22B;(* linked to the EL6001 in the TwinCAT System Manager *)

	Timer		: TON := (PT:=T#0.025S);
	bSendBusy	: BOOL;
	eSendErrorID: ComError_t;

	fbReceive		: ReceiveString;
	sReceivedString	: STRING;
	sLastReceivedString: STRING;
	bStringReceived	: BOOL;
	bReceiveBusy	: BOOL;
	bReceiveError	: BOOL;
	eReceiveErrorID	: ComError_t;
	bReceiveTimeout	: BOOL;
	nReceiveCounter	: UDINT;
	sendErrorStatus: BOOL;
	RcvErrorStatus: BOOL;
	SendPreparedToString: STRING:='M0,0\r';

	arr_SendData : ARRAY [1..20] OF BYTE:=[16#4D, 16#30, 16#2C, 16#30, 16#0D];(*READ*)
	fb_Send: SendData;

	gap_left: LREAL;
	gap_right: LREAL;
END_VAR

(*
The SerialLineControl function block is supposed to be called in every PLC cycle.
It communicates with the serial line hardware device and transmits or receives data.
The SerialLineControl can be called in the standard task (e.g.for PcCOM port usage) 
or in a separate fast task (e.g.for terminal usage) as well.
A fast separate task will be necessary at high baud rates or with KL6001 terminals 
which have a small process image (3 or 5 data bytes only)
*)

(* background communication with the EL6001 terminal *)
fbEL6001Ctrl(
	Mode:= SERIALLINEMODE_KL6_22B_STANDARD,
	pComIn:= ADR(stIn_EL6001),
	pComOut:= ADR(stOut_EL6001),
	SizeComIn:= SIZEOF(stIn_EL6001),
	Error=> ,
	ErrorID=> ,
	TxBuffer:= TxBufferEL,
	RxBuffer:= RxBufferEL );
IF fbEL6001Ctrl.Error THEN
	bEL6001CtrlError := TRUE;
	eEL6001CtrlErrorID := fbEL6001Ctrl.ErrorID;
END_IF

(* Call the send block every second TO REPEAT the transmission.
// Also call the block as long as it is busy to finish a transmission.*)
Timer(IN:=TRUE);
IF Timer.Q OR fb_Send.Busy THEN
	Timer(IN:=FALSE); (* reset timer *)
	sendErrorStatus:=FALSE;
	fb_Send(		pSendData:=ADR(arr_SendData[1]) ,
			Length:=5 ,
			TXbuffer:=TxBufferEL ,
			Busy=>bSendBusy ,
			Error=> );
	IF fb_Send.Error <> COMERROR_NOERROR THEN
		sendErrorStatus:=TRUE;
		eSendErrorID := fb_Send.Error;
	END_IF
END_IF

(*//	Receive string data:
//	The block receives any data strings beginning with a STX ($02) and ending with an ETX ($03) character.	*)
fbReceive(
	(*Prefix:= 'M0,',
	Suffix:= '$R',*)
	Prefix:= ,
	Suffix:= ,
	Timeout:= T#0.025s,
	ReceivedString:= sReceivedString,
	RXbuffer:= RxBufferEL,
	StringReceived=> bStringReceived,
	Busy=> bReceiveBusy,
	Error=> ,
	RxTimeout=> bReceiveTimeout );
IF fbReceive.Error <> COMERROR_NOERROR THEN
	RcvErrorStatus:=TRUE;
	eReceiveErrorID := fbReceive.Error;
ELSE
		RcvErrorStatus:=FALSE;
END_IF
IF bStringReceived THEN
	nReceiveCounter := nReceiveCounter + 1;
	sLastReceivedString := sReceivedString;
END_IF
IF LEN(sLastReceivedString)>=22 THEN
	gap_left:=STRING_TO_LREAL(MID(sLastReceivedString, 9, 4));
	gap_right:=STRING_TO_LREAL(MID(sLastReceivedString, 9, 14));
END_IF

END_PROGRAM
